TEXTLIST LevelTxtList
  1 = 'level [1]'
  2 = 'level [2]'
  3 = 'level [3]'
  4 = 'level [4]'
  5 = 'level [5]'
  6 = 'level [6]'
   = ''
END_TEXTLIST

(* stored: Version 1.1.0.1, ProductVersion 3.1.4022.18
   TextList LevelTxtList: Id {1a00044f-40e8-4b5f-9263-fcc658df7cfc} *)
